Yaskawa INFORM job: BUFFER_INIT.JBI

/JOB
//NAME BUFFER_INIT
//POS
///NPOS 0,0,0,0,0,0
//INST
///DATE 2011/11/29 18:31
///ATTR SC,RW
///GROUP1 RB1
NOP
SET I091 0
SET I092 0
WHILE I092<=I093
ENDWHILE
END
